{attribute addProperty BoxType "EL1512-0000-0016"}
{attribute addProperty Id "CNT_Inputs_ChannelAT %I*ARRAY[0..1] OF CNT_Inputs_Channel_445A37BE128160CNT_Outputs_ChannelAT %Q*ARRAY[0..1] OF CNT_Outputs_Channel_EEA87D4196120WcStateAT %I*WcState_F855686C1620InfoDataAT %I*InfoData_BC63D37F80100"}
{attribute addProperty CRC "1842975781"}
{attribute addProperty SizeInBites "320"}
{attribute addProperty SizeInBytes "40"}
TYPE EL1512_996074CE :
STRUCT
	{attribute addProperty Name "CNT_Inputs_Channel"}
	CNT_Inputs_Channel : ARRAY[0..1] OF CNT_Inputs_Channel_445A37BE;
	{attribute addProperty Name "CNT_Outputs_Channel"}
	CNT_Outputs_Channel : ARRAY[0..1] OF CNT_Outputs_Channel_EEA87D41;
	{attribute addProperty Name "WcState"}
	WcState : WcState_F855686C;
	{attribute addProperty Name "InfoData"}
	InfoData : InfoData_BC63D37F;
END_STRUCT
END_TYPE

(* stored: Version 1.2.0.0, ProductVersion 3.1.4024.9
   DUT EL1512_996074CE: Id {91afd4e2-3a49-475b-8610-0c3c76b7f386} *)
